// TIA Portal V20 export
DATA_BLOCK "DB_LaserAirProcess"   // DB432
// stored: AutoNumber false, InstanceOfName FB_LaserAirProcess, InstanceOfType FB
"FB_LaserAirProcess"
   // VAR
   //    sTimeDelay : Time;
   //    sTimerGas : TON_TIME;
   //    sGasAssistOn : Bool;
   //    sLaser_Air_Process_Ctrl { S7_SetPoint := 'True'} : "FB_AnalogInputThreshold";
   //    sNozzle_Over_Pressure { S7_SetPoint := 'True'} : "FB_AnalogInputThreshold";
   //    sGasAssistDelay { ExternalAccessible := 'False'; ExternalVisible := 'False'; ExternalWritable := 'False'} : Bool;
   //    sGasAssistStartCh1 : Bool;
   //    sGasAssistStartCh2 : Bool;
   //    sGasAssistByKey : Bool;
   //    sGasReadValue : Bool;
   //    sRT_sGasAssistStartCh1 : R_TRIG;
   //    sRT_sGasAssistStartCh2 { S7_SetPoint := 'True'} : R_TRIG;
   //    sFT_sGasAssistStartCh1 { S7_SetPoint := 'True'} : F_TRIG;
   //    sFT_sGasAssistStartCh2 { S7_SetPoint := 'True'} : F_TRIG;
   //    sGasAssistSetPointJog { S7_SetPoint := 'True'} : Real;
   //    sGasAssistOffTimer : TOF_TIME;
   // END_VAR
BEGIN
END_DATA_BLOCK
